KUKA KRL program: collstop.src, collstop.dat

--- collstop.src ---
&ACCESS RVO9
&REL 401
&COMMENT VERRIEGELUNGEN V3.02
DEF  COLLSTOP (NO :IN,MODE :IN )
   ;!======================================================
   ;! Programm : COLLSTOP(..)
   ;! Funktion : Steuerung der Verriegelungen Roboter
   ;!
   ;! Mode 0 = Interruptmodus
   ;! Mode 1 = Einschalten
   ;! Mode 2 = Ausschalten
   ;! Mode 3 = Initialisierung
   ;!
   ;!=======================================================
   ;! Version  : 3.02
   ;! Aenderungsstand: 17.10.01
   ;! (C) 2001 DC-Bremen RBR-IH
   ;! Bearbeiter: Projektgruppe R230 B.S Tel.: 6652
   ;!=======================================================
   ;! Version  : 3.01
   ;! Aenderungsstand: 05.05.2000
   ;!=======================================================
   ;! (C) 1998 Daimler-Benz AG
   ;!
   ;! Bearbeiter: R.Weinmann  07031-90-2571
   ;!=======================================================

   INT NO,MODE,II
   BOOL BRESULT

   SWITCH  MODE

;====main case===========
CASE 0 ;Interruptmodus
;========================
   IF ($EXT) THEN
         SWITCH  NO
         CASE 1
            INTERRUPT DISABLE 21
         CASE 2
            INTERRUPT DISABLE 22
         CASE 3
            INTERRUPT DISABLE 23
         CASE 4
            INTERRUPT DISABLE 24
         DEFAULT
         ENDSWITCH
         BRAKE
         MSG_WAIT ( CS_MESSAGE[], COLLISION_DATA[NO].I_NR,TRUE,MAX_I_CS_MESSAGE, 0,BRESULT )
         SWITCH  NO
         CASE 1
            INTERRUPT ENABLE 21
         CASE 2
            INTERRUPT ENABLE 22
         CASE 3
            INTERRUPT ENABLE 23
         CASE 4
            INTERRUPT ENABLE 24
         DEFAULT
         ENDSWITCH
      ENDIF ;$EXT

;====main case===========
CASE 1 ;Einschalten
;========================
    WHILE  COLLISION_DATA[NO].I_NR==0
         MSG_TEXT (CS_ERRORS[1],#QUIT )
      ENDWHILE
      IF ($EXT) AND (NO<=4) AND (COLLISION_DATA[NO].I_NR>0) THEN
         IF COLLISION_DATA[NO].ACTIVE==TRUE THEN ;Kollision ist aktiv
            COLLISION_DATA[NO].ACTIVE=FALSE
            SWITCH  NO
            CASE 1
               INTERRUPT OFF 21
            CASE 2
               INTERRUPT OFF 22
            CASE 3
               INTERRUPT OFF 23
            CASE 4
               INTERRUPT OFF 24
            DEFAULT
            ENDSWITCH ;NO
         ENDIF
      ENDIF ;$EXT

      IF COLLISION_DATA[NO].I_NR>0 THEN
	IF $OUT[COLLISION_DATA[NO].I_NR]==FALSE then
   	   MSG_WAIT ( CS_MESSAGE[], COLLISION_DATA[NO].I_NR,TRUE,MAX_I_CS_MESSAGE,0, BRESULT )
	ELSE
           $OUT[COLLISION_DATA[NO].I_NR]=TRUE
           MSG_WAIT ( CS_MESSAGE[], COLLISION_DATA[NO].I_NR,FALSE,MAX_I_CS_MESSAGE,0,BRESULT )
           $OUT[COLLISION_DATA[NO].I_NR]=FALSE
        ENDIF
      ENDIF
      IF ($EXT) AND (NO<=4) AND (COLLISION_DATA[NO].I_NR>0) THEN
         COLLISION_DATA[NO].ACTIVE=TRUE
         SWITCH  NO
         CASE 1
            INTERRUPT ON 21
         CASE 2
            INTERRUPT ON 22
         CASE 3
            INTERRUPT ON 23
         CASE 4
            INTERRUPT ON 24
         DEFAULT
         ENDSWITCH ;NO
      ENDIF ;$EXT

      IF COLLISION_DATA[NO].I_NR>0 THEN
         MSG_WAIT ( CS_MESSAGE[], COLLISION_DATA[NO].I_NR,TRUE,MAX_I_CS_MESSAGE,0, BRESULT )
      ENDIF ;

;====main case===========
CASE 2 ;Ausschalten
;========================

      IF COLLISION_DATA[NO].I_NR>0 THEN
         $OUT[COLLISION_DATA[NO].I_NR]=TRUE
      ENDIF ;

      IF ($EXT) AND (NO<=4) AND (COLLISION_DATA[NO].I_NR>0) THEN
         COLLISION_DATA[NO].ACTIVE=FALSE
         SWITCH  NO
         CASE 1
            INTERRUPT OFF 21
         CASE 2
            INTERRUPT OFF 22
         CASE 3
            INTERRUPT OFF 23
         CASE 4
            INTERRUPT OFF 24
         DEFAULT
         ENDSWITCH ;NO
      ENDIF ;$EXT

;====main case===========
CASE 3 ;Initialisierung
;========================

      FOR II=1 TO  MAX_COLL
         IF COLLISION_DATA[II].I_NR>0 THEN
            $OUT[COLLISION_DATA[II].I_NR]=TRUE
            COLLISION_DATA[II].ACTIVE=FALSE
         ENDIF
      ENDFOR

   DEFAULT
   ENDSWITCH ;MODE
END

--- collstop.dat ---
&ACCESS  RVO
&COMMENT VERRIEGELUNGEN V3.02
&REL 400
DEFDAT  COLLSTOP PUBLIC

;FOLD COLLISION_V3.01 ;%{E}
;Achtung: ACTIVE ist nicht projektierbar (28.04.99)
DECL CONST INT MAX_COLL=16
GLOBAL STRUC COLLISIONTYP INT I_NR,BOOL ACTIVE
DECL GLOBAL COLLISIONTYP COLLISION_DATA[16]
COLLISION_DATA[1]={I_NR 864,ACTIVE FALSE}
COLLISION_DATA[2]={I_NR 863,ACTIVE FALSE}
COLLISION_DATA[3]={I_NR 862,ACTIVE FALSE}
COLLISION_DATA[4]={I_NR 861,ACTIVE FALSE}
COLLISION_DATA[5]={I_NR 860,ACTIVE FALSE}
COLLISION_DATA[6]={I_NR 859,ACTIVE FALSE}
COLLISION_DATA[7]={I_NR 858,ACTIVE FALSE}
COLLISION_DATA[8]={I_NR 857,ACTIVE FALSE}
COLLISION_DATA[9]={I_NR 856,ACTIVE FALSE}
COLLISION_DATA[10]={I_NR 855,ACTIVE FALSE}
COLLISION_DATA[11]={I_NR 854,ACTIVE FALSE}
COLLISION_DATA[12]={I_NR 853,ACTIVE FALSE}
COLLISION_DATA[13]={I_NR 852,ACTIVE FALSE}
COLLISION_DATA[14]={I_NR 851,ACTIVE FALSE}
COLLISION_DATA[15]={I_NR 850,ACTIVE FALSE}
COLLISION_DATA[16]={I_NR 849,ACTIVE FALSE}
;ENDFOLD

;FOLD COLLISION_INPUTS_V3.01
INT MAX_I_CS_MESSAGE=32
DECL I_MESSAGETYP CS_MESSAGE[32]
CS_MESSAGE[1]={I_NR 864,I_MSG_TXT[] "08R10E864:Antikollision mit IR 07R10"}
CS_MESSAGE[2]={I_NR 863,I_MSG_TXT[] "08R10E863:Antikollision mit IR 08R20"}
CS_MESSAGE[3]={I_NR 862,I_MSG_TXT[] "08R10E862:Antikollision mit IR 08R20"}
CS_MESSAGE[4]={I_NR 861,I_MSG_TXT[] "08R10E861:Antikollision mit IR 08R30"}
CS_MESSAGE[5]={I_NR 860,I_MSG_TXT[] "XXXXE860:Antikollision mit IR XXXX                          "}
CS_MESSAGE[6]={I_NR 859,I_MSG_TXT[] "XXXXE859:Antikollision mit IR XXXX                          "}
CS_MESSAGE[7]={I_NR 858,I_MSG_TXT[] "XXXXE858:Antikollision mit IR XXXX                          "}
CS_MESSAGE[8]={I_NR 857,I_MSG_TXT[] "XXXXE857:Antikollision mit IR XXXX                          "}
CS_MESSAGE[9]={I_NR 856,I_MSG_TXT[] "XXXXE856:Antikollision mit IR XXXX                          "}
CS_MESSAGE[10]={I_NR 855,I_MSG_TXT[] "XXXXE855:Antikollision mit IR XXXX                          "}
CS_MESSAGE[11]={I_NR 854,I_MSG_TXT[] "XXXXE854:Antikollision mit IR XXXX                          "}
CS_MESSAGE[12]={I_NR 853,I_MSG_TXT[] "XXXXE853:Antikollision mit IR XXXX                          "}
CS_MESSAGE[13]={I_NR 852,I_MSG_TXT[] "XXXXE852:Antikollision mit IR XXXX                          "}
CS_MESSAGE[14]={I_NR 851,I_MSG_TXT[] "XXXXE851:Antikollision mit IR XXXX                          "}
CS_MESSAGE[15]={I_NR 850,I_MSG_TXT[] "XXXXE850:Antikollision mit IR XXXX                          "}
CS_MESSAGE[16]={I_NR 849,I_MSG_TXT[] "XXXXE849:Antikollision mit IR XXXX                          "}
CS_MESSAGE[17]={I_NR 0,I_MSG_TXT[] "XXXXEXXX:Antikollision mit IR XXXX                          "}
CS_MESSAGE[18]={I_NR 0,I_MSG_TXT[] "XXXXEXXX:Antikollision mit IR XXXX                          "}
CS_MESSAGE[19]={I_NR 0,I_MSG_TXT[] "XXXXEXXX:Antikollision mit IR XXXX                          "}
CS_MESSAGE[20]={I_NR 0,I_MSG_TXT[] "XXXXEXXX:Antikollision mit IR XXXX                          "}
CS_MESSAGE[21]={I_NR 0,I_MSG_TXT[] "XXXXEXXX:Antikollision mit IR XXXX                          "}
CS_MESSAGE[22]={I_NR 0,I_MSG_TXT[] "XXXXEXXX:Antikollision mit IR XXXX                          "}
CS_MESSAGE[23]={I_NR 0,I_MSG_TXT[] "XXXXEXXX:Antikollision mit IR XXXX                          "}
CS_MESSAGE[24]={I_NR 0,I_MSG_TXT[] "XXXXEXXX:Antikollision mit IR XXXX                          "}
CS_MESSAGE[25]={I_NR 0,I_MSG_TXT[] "XXXXEXXX:Antikollision mit IR XXXX                          "}
CS_MESSAGE[26]={I_NR 0,I_MSG_TXT[] "XXXXEXXX:Antikollision mit IR XXXX                          "}
CS_MESSAGE[27]={I_NR 0,I_MSG_TXT[] "XXXXEXXX:Antikollision mit IR XXXX                          "}
CS_MESSAGE[28]={I_NR 0,I_MSG_TXT[] "XXXXEXXX:Antikollision mit IR XXXX                          "}
CS_MESSAGE[29]={I_NR 0,I_MSG_TXT[] "XXXXEXXX:Antikollision mit IR XXXX                          "}
CS_MESSAGE[30]={I_NR 0,I_MSG_TXT[] "XXXXEXXX:Antikollision mit IR XXXX                          "}
CS_MESSAGE[31]={I_NR 0,I_MSG_TXT[] "XXXXEXXX:Antikollision mit IR XXXX                          "}
CS_MESSAGE[32]={I_NR 0,I_MSG_TXT[] "Kein Eingangsname projektiert                               "}
;ENDFOLD

;FOLD COLLISION_ERRORS_V3.01
INT MAX_I_CS_ERRORS=8
DECL MSG_TXT_TYP CS_ERRORS[32]
CS_ERRORS[1]={MSGTXT[] "Verriegelungsnummer nicht projektiert                       "}
CS_ERRORS[2]={MSGTXT[] "                                                            "}
CS_ERRORS[3]={MSGTXT[] "                                                            "}
CS_ERRORS[4]={MSGTXT[] "                                                            "}
CS_ERRORS[5]={MSGTXT[] "                                                            "}
CS_ERRORS[6]={MSGTXT[] "                                                            "}
CS_ERRORS[7]={MSGTXT[] "                                                            "}
CS_ERRORS[8]={MSGTXT[] "                                                            "}
;ENDFOLD

ENDDAT
